// TIA Portal V20 export
DATA_BLOCK "Hmi"   // DB75
{ S7_Optimized_Access := 'FALSE'; DB_Accessible_From_OPC_UA := 'FALSE' }
AUTHOR : MICROTEC
FAMILY : HMI
NAME : HMI
VERSION : 1.0
// stored: AutoNumber false, DBAccessibleFromOPCUA false
   VAR RETAIN
      Clock : Struct
         Act : Date_And_Time;
         Tar : Date_And_Time;
         Set : Bool;
         Read : Bool;
      END_STRUCT;
      operatingHours : DInt;   // complete operating hours from Cpu
      TimeOfDay : Time_Of_Day;
      TimeStamp : DTL;
   END_VAR
BEGIN
END_DATA_BLOCK
